TYPE FastAttenuationConfigs :
STRUCT
	Std900FastAttenuationConfig : Std900FastAttenuationConfig;
END_STRUCT
END_TYPE

(* stored: Version 1.1.0.1, ProductVersion 3.1.4024.3
   DUT FastAttenuationConfigs: Id {4894644f-114b-4861-b5de-90f605964915} *)
